PROGRAM PRG_ExtruderSys
VAR
	fbExtrusionSystem: FB_ExtrusionSystem;
END_VAR

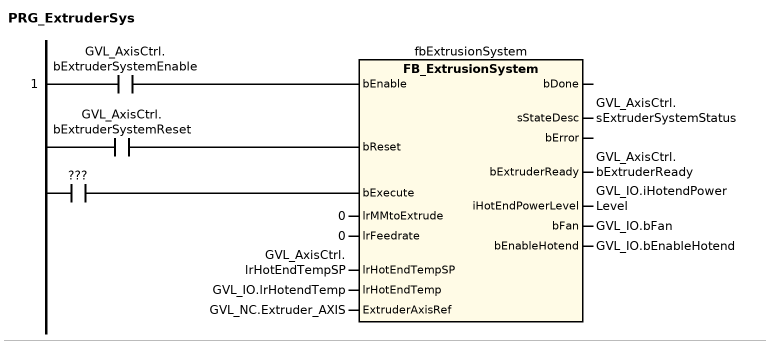
// NETWORK 1
fbExtrusionSystem(
    bEnable := GVL_AxisCtrl.bExtruderSystemEnable,
    bReset := GVL_AxisCtrl.bExtruderSystemReset,
    lrMMtoExtrude := 0,
    lrFeedrate := 0,
    lrHotEndTempSP := GVL_AxisCtrl.lrHotEndTempSP,
    lrHotEndTemp := GVL_IO.lrHotendTemp,
    ExtruderAxisRef := GVL_NC.Extruder_AXIS,
    sStateDesc => GVL_AxisCtrl.sExtruderSystemStatus,
    bExtruderReady => GVL_AxisCtrl.bExtruderReady,
    iHotEndPowerLevel => GVL_IO.iHotendPowerLevel,
    bFan => GVL_IO.bFan,
    bEnableHotend => GVL_IO.bEnableHotend); // FB_ExtrusionSystem

END_PROGRAM

(* stored: Version 1.1.0.1, ProductVersion 3.1.4024.2
   POU PRG_ExtruderSys: Id {7117f760-ae2a-4f57-8081-7475ebd0506e}, SpecialFunc None *)
